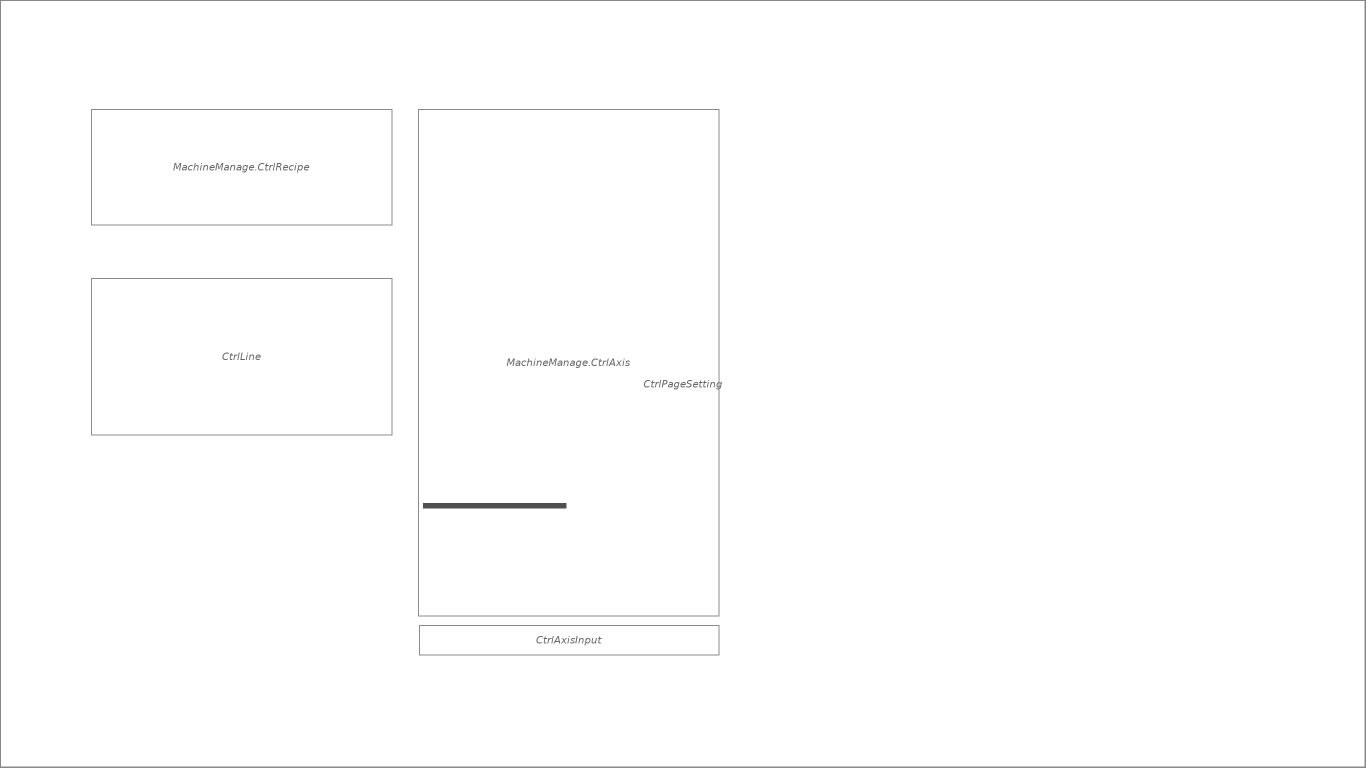
VISUALIZATION PageSetting_Other  // 1366x768
    Frame (0,0 1366x768)
        shows CtrlPageSetting()
    Frame (418,109 301x507)
        shows MachineManage.CtrlAxis(System := G_stSystem, Axis := G_arrAxis[E_Axis.Z], Data := G_arrAxisData[E_Axis.Z])
    Frame (419,625 300x30)
        shows CtrlAxisInput(In := GVL_IO.AxisInput)
    Frame (91,109 301x116)
        shows MachineManage.CtrlRecipe()
    Frame (91,278 301x157)
        shows CtrlLine()
    Rectangle (423,503 143x5), colour toggle: G_arrAxis[E_Axis.Z].Axis_REF.Status.Error OR G_arrAxis[E_Axis.Z].Axis_REF.Status.Disabled
END_VISUALIZATION

(* stored: Version 1.1.0.1, ProductVersion 3.1.4024.3
   Visu PageSetting_Other: Id {a67cfc44-96c0-451d-932d-cfd0862fd22d} *)
